PROGRAM MAIN
VAR
	i: BYTE := 0;
	bStart: BOOL := TRUE;
	bLog: BOOL := FALSE;

	//Query Builder for Document DB
	fbNoSqlQueryBuilder_DocumentDB: FB_NoSQLQueryBuilder_DocumentDB;
	InsertQueryOption: T_QueryOptionDocumentDB_Insert;
	sDocument: STRING (1000);

	//Query Execution
	fbNoSqlQuery: FB_NoSQLQueryEvt(sNetID:= '', tTimeout:= T#5S);
	myDBID: UDINT := 1;
	TcMessage: I_TcMessage;
END_VAR

IF bStart THEN
	CreateQuery();
	bStart:= FALSE;
END_IF

IF bLog THEN
	CreateDocument();
	IF fbNoSqlQuery.Execute(hDBID:= myDBID, iNoSQLQueryBuilder:= fbNoSqlQueryBuilder_DocumentDB) THEN
		IF fbNoSqlQuery.bError THEN
			TcMessage:= fbNoSqlQuery.ipTcResult;
		END_IF
		bLog:= FALSE;
		i := i + 1;
	END_IF
END_IF

ACTION CreateDocument:
sDocument:= '{"name": "son",
				"position": "intern",
				"dateOfBirth": "27-07-1999",
				"number":';
sDocument := CONCAT(STR1:= sDocument, STR2:= BYTE_TO_STRING(i));
sDocument := CONCAT(STR1:= sDocument, STR2:= '}');
END_ACTION

ACTION CreateQuery:
InsertQueryOption.pDocuments := ADR(sDocument);
InsertQueryOption.cbDocuments := SIZEOF(sDocument);

fbNoSqlQueryBuilder_DocumentDB.eQueryType := E_DocumentDbQueryType.InsertOne;
fbNoSqlQueryBuilder_DocumentDB.sCollectionName := 'Customer';
fbNoSqlQueryBuilder_DocumentDB.pQueryOptions := ADR(InsertQueryOption);
fbNoSqlQueryBuilder_DocumentDB.cbQueryOptions := SIZEOF(InsertQueryOption);
END_ACTION

END_PROGRAM

(* stored: Version 1.1.0.1, ProductVersion 3.1.4024.4
   POU MAIN: Id {739b46bf-d99f-41e1-a248-f35519a17b2d}, SpecialFunc None
   Action CreateDocument: Id {bb4591cd-873d-4799-aa4b-b85a07d5e57e}
   Action CreateQuery: Id {2655315e-f323-4ad5-bfc9-07379b6667a2} *)
